// TIA Portal V20 export
DATA_BLOCK "Config"   // DB60
{ DB_Accessible_From_OPC_UA := 'FALSE' }
AUTHOR : ERsystem_FA2_DH. Kim
// stored: Access Published, DBAccessibleFromOPCUA false, DBAccessibleFromWebserver false, MemoryReserve 100, Namespace Unit1.Em4
   VAR RETAIN
      em { ExternalWritable := 'False'} : "LAF_typeEmConfiguration";
      axis { ExternalAccessible := 'False'; ExternalVisible := 'False'; ExternalWritable := 'False'} : Array[1.._.U1EM4_NO_OF_AXES] of DB_ANY;
      cam { ExternalAccessible := 'False'; ExternalVisible := 'False'; ExternalWritable := 'False'} : Array[1.._.U1EM4_NO_OF_CAM] of DB_ANY;
      outputCam { ExternalAccessible := 'False'; ExternalVisible := 'False'; ExternalWritable := 'False'} : Array[1.._.U1EM4_NO_OF_OUTPUTCAM] of DB_ANY;
      cmPnp1stAnodeDetect { S7_SetPoint := 'True'} : "LBC_typeDigitalSignalConfiguration";
      cmPnp2ndAnodeDetect { S7_SetPoint := 'True'} : "LBC_typeDigitalSignalConfiguration";
      cmAnodeAlignTableElectrodeDetect { S7_SetPoint := 'True'} : "LBC_typeDigitalSignalConfiguration";
      cmAnodeNgPnpElectrodeDetect { S7_SetPoint := 'True'} : "LBC_typeDigitalSignalConfiguration";
      cmAnodeNgBoxFullSensorDetect { S7_SetPoint := 'True'} : "LBC_typeDigitalSignalConfiguration";
      cmAnodeNgBoxDetect { S7_SetPoint := 'True'} : "LBC_typeDigitalSignalConfiguration";
      cmAnodeMainPnP1AxisX { ExternalAccessible := 'False'; ExternalVisible := 'False'; ExternalWritable := 'False'} : "LBC_typeAxis64PosConfiguration";
      cmAnodeMainPnP1AxisY { ExternalAccessible := 'False'; ExternalVisible := 'False'; ExternalWritable := 'False'} : "LBC_typeAxis64PosConfiguration";
      cmAnodeMainPnP1AxisZ { ExternalAccessible := 'False'; ExternalVisible := 'False'; ExternalWritable := 'False'} : "LBC_typeAxis64PosConfiguration";
      cmAnodeMainPnP2AxisX { ExternalAccessible := 'False'; ExternalVisible := 'False'; ExternalWritable := 'False'} : "LBC_typeAxis64PosConfiguration";
      cmAnodeMainPnP2AxisZ { ExternalAccessible := 'False'; ExternalVisible := 'False'; ExternalWritable := 'False'} : "LBC_typeAxis64PosConfiguration";
      cmAnodeAlignTableAxisX { ExternalAccessible := 'False'; ExternalVisible := 'False'; ExternalWritable := 'False'} : "LBC_typeAxis64PosConfiguration";
      cmAnodeAlignTableAxisY1 { ExternalAccessible := 'False'; ExternalVisible := 'False'; ExternalWritable := 'False'} : "LBC_typeAxis64PosConfiguration";
      cmAnodeAlignTableAxisY2 { ExternalAccessible := 'False'; ExternalVisible := 'False'; ExternalWritable := 'False'} : "LBC_typeAxis64PosConfiguration";
      cmAnodeMainPnP1RotaryCwCcw { ExternalAccessible := 'False'; ExternalVisible := 'False'; ExternalWritable := 'False'} : "LBC_typeTwoWayActuatorConfiguration";
      cmAnodeMainPnP1SuctionPlateVacuum { ExternalAccessible := 'False'; ExternalVisible := 'False'; ExternalWritable := 'False'} : "LBC_typeTwoWayActuatorConfiguration";
      cmAnodeMainPnP2SuctionPlateVacuum { ExternalAccessible := 'False'; ExternalVisible := 'False'; ExternalWritable := 'False'} : "LBC_typeTwoWayActuatorConfiguration";
      cmAnodeAlignTableSuctionPlateVacuum { ExternalAccessible := 'False'; ExternalVisible := 'False'; ExternalWritable := 'False'} : "LBC_typeTwoWayActuatorConfiguration";
      cmAnodeGlassCleaning { ExternalAccessible := 'False'; ExternalVisible := 'False'; ExternalWritable := 'False'} : "LBC_typeTwoWayActuatorConfiguration";
      cmAnodeNgPnpUpDown { ExternalAccessible := 'False'; ExternalVisible := 'False'; ExternalWritable := 'False'} : "LBC_typeTwoWayActuatorConfiguration";
      cmAnodeNgPnp1stFwdBwd { ExternalAccessible := 'False'; ExternalVisible := 'False'; ExternalWritable := 'False'; S7_SetPoint := 'True'} : "LBC_typeTwoWayActuatorConfiguration";
      cmAnodeNgPnp2ndFwdBwd { ExternalAccessible := 'False'; ExternalVisible := 'False'; ExternalWritable := 'False'; S7_SetPoint := 'True'} : "LBC_typeTwoWayActuatorConfiguration";
      cmAnodeMaintenanceMovingFixFrontRearFwdBwd { ExternalAccessible := 'False'; ExternalVisible := 'False'; ExternalWritable := 'False'} : "LBC_typeTwoWayActuatorConfiguration";
      cmAnodeNgBoxLiftUpDown { ExternalAccessible := 'False'; ExternalVisible := 'False'; ExternalWritable := 'False'; S7_SetPoint := 'True'} : "LBC_typeTwoWayActuatorConfiguration";
      cmAnodeNgBoxLockUpDown { ExternalAccessible := 'False'; ExternalVisible := 'False'; ExternalWritable := 'False'; S7_SetPoint := 'True'} : "LBC_typeTwoWayActuatorConfiguration";
      cmAnodeNgPnpVaccum { ExternalAccessible := 'False'; ExternalVisible := 'False'; ExternalWritable := 'False'; S7_SetPoint := 'True'} : "LBC_typeTwoWayActuatorConfiguration";
      cmAnodeConveyorCoverFwdBwd { S7_SetPoint := 'True'} : "LBC_typeTwoWayActuatorConfiguration";
      cmAnodeConveyorPickUpBlower { S7_SetPoint := 'True'} : "LBC_typeTwoWayActuatorConfiguration";
      cmAnodeVisionControllerInterface { ExternalAccessible := 'False'; ExternalVisible := 'False'; ExternalWritable := 'False'} : "LER_typeVisionConfiguration";
      softCam : Struct
         cmAnodeMainPnP1AxisX : "LER_typeSoftCamInterface";
         cmAnodeMainPnP1AxisY { S7_SetPoint := 'True'} : "LER_typeSoftCamInterface";
         cmAnodeMainPnP1AxisZ { S7_SetPoint := 'True'} : "LER_typeSoftCamInterface";
         cmAnodeMainPnP2AxisX { S7_SetPoint := 'True'} : "LER_typeSoftCamInterface";
         cmAnodeMainPnP2AxisZ { S7_SetPoint := 'True'} : "LER_typeSoftCamInterface";
         cmAnodeAlignTableAxisX { S7_SetPoint := 'True'} : "LER_typeSoftCamInterface";
         cmAnodeAlignTableAxisY1 { S7_SetPoint := 'True'} : "LER_typeSoftCamInterface";
         cmAnodeAlignTableAxisY2 { S7_SetPoint := 'True'} : "LER_typeSoftCamInterface";
      END_STRUCT;
   END_VAR
BEGIN
   em.referenceDesignator.parent := WSTRING#'';
   em.referenceDesignator.relative := WSTRING#'';
   em.referenceDesignator.combined := WSTRING#'';
   axis[1] := 144;   // AnodeMainPnP1AxisX
   axis[2] := 145;   // AnodeMainPnP2AxisX
   axis[3] := 148;   // AnodeMainPnP1AxisY
   axis[4] := 149;   // AnodeMainPnP1AxisZ
   axis[5] := 150;   // AnodeMainPnP2AxisZ
   axis[6] := 154;   // AnodeAlignTableAxisX
   axis[7] := 155;   // AnodeAlignTableAxisY1
   axis[8] := 156;   // AnodeAlignTableAxisY2
   cam[1] := 144;   // AnodeMainPnP1AxisX
   cam[2] := 145;   // AnodeMainPnP2AxisX
   cam[3] := 148;   // AnodeMainPnP1AxisY
   cam[4] := 149;   // AnodeMainPnP1AxisZ
   outputCam[1] := 412;
   outputCam[2] := 413;
   outputCam[3] := 414;
   outputCam[4] := 415;
   outputCam[5] := 441;
   outputCam[6] := 420;
   outputCam[7] := 437;
   outputCam[8] := 438;
   outputCam[9] := 430;
   outputCam[10] := 432;
   outputCam[11] := 436;
   outputCam[12] := 434;
   outputCam[13] := 433;
   outputCam[14] := 431;
   outputCam[15] := 185;
   outputCam[16] := 435;
   outputCam[17] := 442;
   outputCam[18] := 455;
   outputCam[19] := 456;
   outputCam[20] := 134;
   outputCam[21] := 140;
   outputCam[22] := 187;
   cmPnp1stAnodeDetect.referenceDesignator := WSTRING#'Pnp1stAnodeDetect';
   cmPnp1stAnodeDetect.onDelay := T#0MS;
   cmPnp1stAnodeDetect.offDelay := T#0MS;
   cmPnp1stAnodeDetect.default := FALSE;
   cmPnp1stAnodeDetect.invertProcessValue := FALSE;
   cmPnp1stAnodeDetect.disableAlarms := FALSE;
   cmPnp2ndAnodeDetect.referenceDesignator := WSTRING#'Pnp2ndAnodeDetect';
   cmPnp2ndAnodeDetect.onDelay := T#0MS;
   cmPnp2ndAnodeDetect.offDelay := T#0MS;
   cmPnp2ndAnodeDetect.default := FALSE;
   cmPnp2ndAnodeDetect.invertProcessValue := FALSE;
   cmPnp2ndAnodeDetect.disableAlarms := FALSE;
   cmAnodeAlignTableElectrodeDetect.referenceDesignator := WSTRING#'AlignTableElectrodeDetect';
   cmAnodeAlignTableElectrodeDetect.onDelay := T#0MS;
   cmAnodeAlignTableElectrodeDetect.offDelay := T#0MS;
   cmAnodeAlignTableElectrodeDetect.default := FALSE;
   cmAnodeAlignTableElectrodeDetect.invertProcessValue := FALSE;
   cmAnodeAlignTableElectrodeDetect.disableAlarms := FALSE;
   cmAnodeNgPnpElectrodeDetect.referenceDesignator := WSTRING#'NgPnpElectrodeDetect';
   cmAnodeNgPnpElectrodeDetect.onDelay := T#0MS;
   cmAnodeNgPnpElectrodeDetect.offDelay := T#0MS;
   cmAnodeNgPnpElectrodeDetect.default := FALSE;
   cmAnodeNgPnpElectrodeDetect.invertProcessValue := FALSE;
   cmAnodeNgPnpElectrodeDetect.disableAlarms := FALSE;
   cmAnodeNgBoxFullSensorDetect.referenceDesignator := WSTRING#'NgBoxFullSensorDetect';
   cmAnodeNgBoxFullSensorDetect.onDelay := T#0MS;
   cmAnodeNgBoxFullSensorDetect.offDelay := T#0MS;
   cmAnodeNgBoxFullSensorDetect.default := FALSE;
   cmAnodeNgBoxFullSensorDetect.invertProcessValue := FALSE;
   cmAnodeNgBoxFullSensorDetect.disableAlarms := FALSE;
   cmAnodeNgBoxDetect.referenceDesignator := WSTRING#'NgBoxDetect';
   cmAnodeNgBoxDetect.onDelay := T#0MS;
   cmAnodeNgBoxDetect.offDelay := T#0MS;
   cmAnodeNgBoxDetect.default := FALSE;
   cmAnodeNgBoxDetect.invertProcessValue := FALSE;
   cmAnodeNgBoxDetect.disableAlarms := FALSE;
   cmAnodeMainPnP1AxisX.referenceDesignator := WSTRING#'AnodeMainPnP1AxisX';
   cmAnodeMainPnP1AxisX.disableAlarms := FALSE;
   cmAnodeMainPnP1AxisX.masterControlPopUp := TRUE;
   cmAnodeMainPnP1AxisX.setPositions[0].position := 540.0;
   cmAnodeMainPnP1AxisX.setPositions[1].position := 0.0;
   cmAnodeMainPnP1AxisX.setPositions[2].position := -5.0;
   cmAnodeMainPnP1AxisX.setPositions[3..15].position := 0.0;
   cmAnodeMainPnP1AxisX.setPositions[0..1].velocity := 500.0;
   cmAnodeMainPnP1AxisX.setPositions[2..3].velocity := 1040.0;
   cmAnodeMainPnP1AxisX.setPositions[4..15].velocity := -1.0;
   cmAnodeMainPnP1AxisX.setPositions[0..1].acceleration := 5000.0;
   cmAnodeMainPnP1AxisX.setPositions[2..3].acceleration := 10400.0;
   cmAnodeMainPnP1AxisX.setPositions[4..15].acceleration := -1.0;
   cmAnodeMainPnP1AxisX.setPositions[0..1].deceleration := 5000.0;
   cmAnodeMainPnP1AxisX.setPositions[2..3].deceleration := 10400.0;
   cmAnodeMainPnP1AxisX.setPositions[4..15].deceleration := -1.0;
   cmAnodeMainPnP1AxisX.setPositions[0..15]."name" := '';
   cmAnodeMainPnP1AxisY.referenceDesignator := WSTRING#'AnodeMainPnP1AxisY';
   cmAnodeMainPnP1AxisY.disableAlarms := FALSE;
   cmAnodeMainPnP1AxisY.masterControlPopUp := TRUE;
   cmAnodeMainPnP1AxisY.setPositions[0..15].position := 0.0;
   cmAnodeMainPnP1AxisY.setPositions[0].velocity := 50.0;
   cmAnodeMainPnP1AxisY.setPositions[1].velocity := 30.0;
   cmAnodeMainPnP1AxisY.setPositions[2..15].velocity := -1.0;
   cmAnodeMainPnP1AxisY.setPositions[0].acceleration := 500.0;
   cmAnodeMainPnP1AxisY.setPositions[1].acceleration := 30.0;
   cmAnodeMainPnP1AxisY.setPositions[2..15].acceleration := -1.0;
   cmAnodeMainPnP1AxisY.setPositions[0].deceleration := 500.0;
   cmAnodeMainPnP1AxisY.setPositions[1].deceleration := 30.0;
   cmAnodeMainPnP1AxisY.setPositions[2..15].deceleration := -1.0;
   cmAnodeMainPnP1AxisY.setPositions[0..15]."name" := '';
   cmAnodeMainPnP1AxisZ.referenceDesignator := WSTRING#'AnodeMainPnP1AxisZ';
   cmAnodeMainPnP1AxisZ.disableAlarms := FALSE;
   cmAnodeMainPnP1AxisZ.masterControlPopUp := TRUE;
   cmAnodeMainPnP1AxisZ.setPositions[0].position := 0.0;
   cmAnodeMainPnP1AxisZ.setPositions[1].position := 20.0;
   cmAnodeMainPnP1AxisZ.setPositions[2..3].position := 30.0;
   cmAnodeMainPnP1AxisZ.setPositions[4..15].position := 0.0;
   cmAnodeMainPnP1AxisZ.setPositions[0..3].velocity := 50.0;
   cmAnodeMainPnP1AxisZ.setPositions[4..15].velocity := -1.0;
   cmAnodeMainPnP1AxisZ.setPositions[0..3].acceleration := 500.0;
   cmAnodeMainPnP1AxisZ.setPositions[4..15].acceleration := -1.0;
   cmAnodeMainPnP1AxisZ.setPositions[0..3].deceleration := 500.0;
   cmAnodeMainPnP1AxisZ.setPositions[4..15].deceleration := -1.0;
   cmAnodeMainPnP1AxisZ.setPositions[0..15]."name" := '';
   cmAnodeMainPnP2AxisX.referenceDesignator := WSTRING#'AnodeMainPnP2AxisX';
   cmAnodeMainPnP2AxisX.disableAlarms := FALSE;
   cmAnodeMainPnP2AxisX.masterControlPopUp := TRUE;
   cmAnodeMainPnP2AxisX.setPositions[0].position := 540.0;
   cmAnodeMainPnP2AxisX.setPositions[1].position := 0.0;
   cmAnodeMainPnP2AxisX.setPositions[2].position := -3.5;
   cmAnodeMainPnP2AxisX.setPositions[3..15].position := 0.0;
   cmAnodeMainPnP2AxisX.setPositions[0..1].velocity := 500.0;
   cmAnodeMainPnP2AxisX.setPositions[2..3].velocity := 1040.0;
   cmAnodeMainPnP2AxisX.setPositions[4..15].velocity := -1.0;
   cmAnodeMainPnP2AxisX.setPositions[0..1].acceleration := 5000.0;
   cmAnodeMainPnP2AxisX.setPositions[2..3].acceleration := 10400.0;
   cmAnodeMainPnP2AxisX.setPositions[4..15].acceleration := -1.0;
   cmAnodeMainPnP2AxisX.setPositions[0..1].deceleration := 5000.0;
   cmAnodeMainPnP2AxisX.setPositions[2..3].deceleration := 10400.0;
   cmAnodeMainPnP2AxisX.setPositions[4..15].deceleration := -1.0;
   cmAnodeMainPnP2AxisX.setPositions[0..15]."name" := '';
   cmAnodeMainPnP2AxisZ.referenceDesignator := WSTRING#'AnodeMainPnP2AxisZ';
   cmAnodeMainPnP2AxisZ.disableAlarms := FALSE;
   cmAnodeMainPnP2AxisZ.masterControlPopUp := TRUE;
   cmAnodeMainPnP2AxisZ.setPositions[0].position := 0.0;
   cmAnodeMainPnP2AxisZ.setPositions[1].position := 20.0;
   cmAnodeMainPnP2AxisZ.setPositions[2..3].position := 30.0;
   cmAnodeMainPnP2AxisZ.setPositions[4..15].position := 0.0;
   cmAnodeMainPnP2AxisZ.setPositions[0..3].velocity := 50.0;
   cmAnodeMainPnP2AxisZ.setPositions[4..15].velocity := -1.0;
   cmAnodeMainPnP2AxisZ.setPositions[0..3].acceleration := 500.0;
   cmAnodeMainPnP2AxisZ.setPositions[4..15].acceleration := -1.0;
   cmAnodeMainPnP2AxisZ.setPositions[0..3].deceleration := 500.0;
   cmAnodeMainPnP2AxisZ.setPositions[4..15].deceleration := -1.0;
   cmAnodeMainPnP2AxisZ.setPositions[0..15]."name" := '';
   cmAnodeAlignTableAxisX.referenceDesignator := WSTRING#'AnodeAlignTableAxisX';
   cmAnodeAlignTableAxisX.disableAlarms := FALSE;
   cmAnodeAlignTableAxisX.masterControlPopUp := TRUE;
   cmAnodeAlignTableAxisX.setPositions[0].position := 0.0;
   cmAnodeAlignTableAxisX.setPositions[1].position := 1.0;
   cmAnodeAlignTableAxisX.setPositions[2..3].position := -4.08;
   cmAnodeAlignTableAxisX.setPositions[4].position := -2.08;
   cmAnodeAlignTableAxisX.setPositions[5..7].position := -0.08;
   cmAnodeAlignTableAxisX.setPositions[8].position := -2.08;
   cmAnodeAlignTableAxisX.setPositions[9].position := -4.08;
   cmAnodeAlignTableAxisX.setPositions[10].position := 8.5;
   cmAnodeAlignTableAxisX.setPositions[11..15].position := 0.0;
   cmAnodeAlignTableAxisX.setPositions[0..1].velocity := 50.0;
   cmAnodeAlignTableAxisX.setPositions[2..9].velocity := 30.0;
   cmAnodeAlignTableAxisX.setPositions[10..15].velocity := -1.0;
   cmAnodeAlignTableAxisX.setPositions[0..1].acceleration := 500.0;
   cmAnodeAlignTableAxisX.setPositions[2..9].acceleration := 30.0;
   cmAnodeAlignTableAxisX.setPositions[10..15].acceleration := -1.0;
   cmAnodeAlignTableAxisX.setPositions[0..1].deceleration := 500.0;
   cmAnodeAlignTableAxisX.setPositions[2..9].deceleration := 30.0;
   cmAnodeAlignTableAxisX.setPositions[10..15].deceleration := -1.0;
   cmAnodeAlignTableAxisX.setPositions[0..15]."name" := '';
   cmAnodeAlignTableAxisY1.referenceDesignator := WSTRING#'AnodeAlignTableAxisY1';
   cmAnodeAlignTableAxisY1.disableAlarms := FALSE;
   cmAnodeAlignTableAxisY1.masterControlPopUp := TRUE;
   cmAnodeAlignTableAxisY1.setPositions[0].position := 0.0;
   cmAnodeAlignTableAxisY1.setPositions[1].position := 2.0;
   cmAnodeAlignTableAxisY1.setPositions[2].position := 0.6;
   cmAnodeAlignTableAxisY1.setPositions[3..5].position := 2.6;
   cmAnodeAlignTableAxisY1.setPositions[6].position := 0.6;
   cmAnodeAlignTableAxisY1.setPositions[7].position := -1.4;
   cmAnodeAlignTableAxisY1.setPositions[8].position := 0.6;
   cmAnodeAlignTableAxisY1.setPositions[9].position := -1.4;
   cmAnodeAlignTableAxisY1.setPositions[10].position := 8.5;
   cmAnodeAlignTableAxisY1.setPositions[11..15].position := 0.0;
   cmAnodeAlignTableAxisY1.setPositions[0..1].velocity := 50.0;
   cmAnodeAlignTableAxisY1.setPositions[2..9].velocity := 30.0;
   cmAnodeAlignTableAxisY1.setPositions[10..15].velocity := -1.0;
   cmAnodeAlignTableAxisY1.setPositions[0..1].acceleration := 500.0;
   cmAnodeAlignTableAxisY1.setPositions[2..9].acceleration := 30.0;
   cmAnodeAlignTableAxisY1.setPositions[10..15].acceleration := -1.0;
   cmAnodeAlignTableAxisY1.setPositions[0..1].deceleration := 500.0;
   cmAnodeAlignTableAxisY1.setPositions[2..9].deceleration := 30.0;
   cmAnodeAlignTableAxisY1.setPositions[10..15].deceleration := -1.0;
   cmAnodeAlignTableAxisY1.setPositions[0..15]."name" := '';
   cmAnodeAlignTableAxisY2.referenceDesignator := WSTRING#'AnodeAlignTableAxisY2';
   cmAnodeAlignTableAxisY2.disableAlarms := FALSE;
   cmAnodeAlignTableAxisY2.masterControlPopUp := TRUE;
   cmAnodeAlignTableAxisY2.setPositions[0].position := 0.0;
   cmAnodeAlignTableAxisY2.setPositions[1].position := 3.0;
   cmAnodeAlignTableAxisY2.setPositions[2..9].position := 0.0;
   cmAnodeAlignTableAxisY2.setPositions[10].position := 8.5;
   cmAnodeAlignTableAxisY2.setPositions[11..15].position := 0.0;
   cmAnodeAlignTableAxisY2.setPositions[0..1].velocity := 50.0;
   cmAnodeAlignTableAxisY2.setPositions[2..15].velocity := -1.0;
   cmAnodeAlignTableAxisY2.setPositions[0..1].acceleration := 500.0;
   cmAnodeAlignTableAxisY2.setPositions[2..15].acceleration := -1.0;
   cmAnodeAlignTableAxisY2.setPositions[0..1].deceleration := 500.0;
   cmAnodeAlignTableAxisY2.setPositions[2..15].deceleration := -1.0;
   cmAnodeAlignTableAxisY2.setPositions[0..15]."name" := '';
   cmAnodeMainPnP1RotaryCwCcw.monitoringLeavingFeedback := T#1S;
   cmAnodeMainPnP1RotaryCwCcw.monitoringReachingFeedback := T#1S;
   cmAnodeMainPnP1RotaryCwCcw.monitoringDiscrepancy := T#0MS;
   cmAnodeMainPnP1RotaryCwCcw.setOutputHomeContinuously := TRUE;
   cmAnodeMainPnP1RotaryCwCcw.setOutputWorkContinuously := TRUE;
   cmAnodeMainPnP1RotaryCwCcw.disableHomeCommand := FALSE;
   cmAnodeMainPnP1RotaryCwCcw.disableFeedbackHomePos := TRUE;
   cmAnodeMainPnP1RotaryCwCcw.disableFeedbackWorkPos := TRUE;
   cmAnodeMainPnP1RotaryCwCcw.disableAlarms := TRUE;
   cmAnodeMainPnP1RotaryCwCcw.resetOutputsOnError := FALSE;
   cmAnodeMainPnP1RotaryCwCcw.allwaysWaitOnReachingTime := FALSE;
   cmAnodeMainPnP1SuctionPlateVacuum.monitoringLeavingFeedback := T#1S;
   cmAnodeMainPnP1SuctionPlateVacuum.monitoringReachingFeedback := T#1S;
   cmAnodeMainPnP1SuctionPlateVacuum.monitoringDiscrepancy := T#15S;
   cmAnodeMainPnP1SuctionPlateVacuum.setOutputHomeContinuously := TRUE;
   cmAnodeMainPnP1SuctionPlateVacuum.setOutputWorkContinuously := TRUE;
   cmAnodeMainPnP1SuctionPlateVacuum.disableHomeCommand := FALSE;
   cmAnodeMainPnP1SuctionPlateVacuum.disableFeedbackHomePos := FALSE;
   cmAnodeMainPnP1SuctionPlateVacuum.disableFeedbackWorkPos := FALSE;
   cmAnodeMainPnP1SuctionPlateVacuum.disableAlarms := FALSE;
   cmAnodeMainPnP1SuctionPlateVacuum.resetOutputsOnError := FALSE;
   cmAnodeMainPnP1SuctionPlateVacuum.allwaysWaitOnReachingTime := FALSE;
   cmAnodeMainPnP2SuctionPlateVacuum.monitoringLeavingFeedback := T#1S;
   cmAnodeMainPnP2SuctionPlateVacuum.monitoringReachingFeedback := T#1S;
   cmAnodeMainPnP2SuctionPlateVacuum.monitoringDiscrepancy := T#15S;
   cmAnodeMainPnP2SuctionPlateVacuum.setOutputHomeContinuously := TRUE;
   cmAnodeMainPnP2SuctionPlateVacuum.setOutputWorkContinuously := TRUE;
   cmAnodeMainPnP2SuctionPlateVacuum.disableHomeCommand := FALSE;
   cmAnodeMainPnP2SuctionPlateVacuum.disableFeedbackHomePos := FALSE;
   cmAnodeMainPnP2SuctionPlateVacuum.disableFeedbackWorkPos := FALSE;
   cmAnodeMainPnP2SuctionPlateVacuum.disableAlarms := FALSE;
   cmAnodeMainPnP2SuctionPlateVacuum.resetOutputsOnError := FALSE;
   cmAnodeMainPnP2SuctionPlateVacuum.allwaysWaitOnReachingTime := FALSE;
   cmAnodeAlignTableSuctionPlateVacuum.monitoringLeavingFeedback := T#1S;
   cmAnodeAlignTableSuctionPlateVacuum.monitoringReachingFeedback := T#1S;
   cmAnodeAlignTableSuctionPlateVacuum.monitoringDiscrepancy := T#0MS;
   cmAnodeAlignTableSuctionPlateVacuum.setOutputHomeContinuously := TRUE;
   cmAnodeAlignTableSuctionPlateVacuum.setOutputWorkContinuously := TRUE;
   cmAnodeAlignTableSuctionPlateVacuum.disableHomeCommand := FALSE;
   cmAnodeAlignTableSuctionPlateVacuum.disableFeedbackHomePos := FALSE;
   cmAnodeAlignTableSuctionPlateVacuum.disableFeedbackWorkPos := FALSE;
   cmAnodeAlignTableSuctionPlateVacuum.disableAlarms := FALSE;
   cmAnodeAlignTableSuctionPlateVacuum.resetOutputsOnError := FALSE;
   cmAnodeAlignTableSuctionPlateVacuum.allwaysWaitOnReachingTime := FALSE;
   cmAnodeGlassCleaning.monitoringLeavingFeedback := T#1S;
   cmAnodeGlassCleaning.monitoringReachingFeedback := T#1S;
   cmAnodeGlassCleaning.monitoringDiscrepancy := T#0MS;
   cmAnodeGlassCleaning.setOutputHomeContinuously := TRUE;
   cmAnodeGlassCleaning.setOutputWorkContinuously := TRUE;
   cmAnodeGlassCleaning.disableHomeCommand := FALSE;
   cmAnodeGlassCleaning.disableFeedbackHomePos := TRUE;
   cmAnodeGlassCleaning.disableFeedbackWorkPos := TRUE;
   cmAnodeGlassCleaning.disableAlarms := FALSE;
   cmAnodeGlassCleaning.resetOutputsOnError := FALSE;
   cmAnodeGlassCleaning.allwaysWaitOnReachingTime := FALSE;
   cmAnodeNgPnpUpDown.monitoringLeavingFeedback := T#5S;
   cmAnodeNgPnpUpDown.monitoringReachingFeedback := T#5S;
   cmAnodeNgPnpUpDown.monitoringDiscrepancy := T#0MS;
   cmAnodeNgPnpUpDown.setOutputHomeContinuously := TRUE;
   cmAnodeNgPnpUpDown.setOutputWorkContinuously := TRUE;
   cmAnodeNgPnpUpDown.disableHomeCommand := FALSE;
   cmAnodeNgPnpUpDown.disableFeedbackHomePos := TRUE;
   cmAnodeNgPnpUpDown.disableFeedbackWorkPos := TRUE;
   cmAnodeNgPnpUpDown.disableAlarms := FALSE;
   cmAnodeNgPnpUpDown.resetOutputsOnError := FALSE;
   cmAnodeNgPnpUpDown.allwaysWaitOnReachingTime := FALSE;
   cmAnodeNgPnp1stFwdBwd.monitoringLeavingFeedback := T#5S;
   cmAnodeNgPnp1stFwdBwd.monitoringReachingFeedback := T#5S;
   cmAnodeNgPnp1stFwdBwd.monitoringDiscrepancy := T#0MS;
   cmAnodeNgPnp1stFwdBwd.setOutputHomeContinuously := TRUE;
   cmAnodeNgPnp1stFwdBwd.setOutputWorkContinuously := TRUE;
   cmAnodeNgPnp1stFwdBwd.disableHomeCommand := FALSE;
   cmAnodeNgPnp1stFwdBwd.disableFeedbackHomePos := TRUE;
   cmAnodeNgPnp1stFwdBwd.disableFeedbackWorkPos := TRUE;
   cmAnodeNgPnp1stFwdBwd.disableAlarms := FALSE;
   cmAnodeNgPnp1stFwdBwd.resetOutputsOnError := FALSE;
   cmAnodeNgPnp1stFwdBwd.allwaysWaitOnReachingTime := FALSE;
   cmAnodeNgPnp2ndFwdBwd.monitoringLeavingFeedback := T#0MS;
   cmAnodeNgPnp2ndFwdBwd.monitoringReachingFeedback := T#0MS;
   cmAnodeNgPnp2ndFwdBwd.monitoringDiscrepancy := T#0MS;
   cmAnodeNgPnp2ndFwdBwd.setOutputHomeContinuously := FALSE;
   cmAnodeNgPnp2ndFwdBwd.setOutputWorkContinuously := FALSE;
   cmAnodeNgPnp2ndFwdBwd.disableHomeCommand := FALSE;
   cmAnodeNgPnp2ndFwdBwd.disableFeedbackHomePos := TRUE;
   cmAnodeNgPnp2ndFwdBwd.disableFeedbackWorkPos := TRUE;
   cmAnodeNgPnp2ndFwdBwd.disableAlarms := FALSE;
   cmAnodeNgPnp2ndFwdBwd.resetOutputsOnError := FALSE;
   cmAnodeNgPnp2ndFwdBwd.allwaysWaitOnReachingTime := FALSE;
   cmAnodeMaintenanceMovingFixFrontRearFwdBwd.monitoringLeavingFeedback := T#5S;
   cmAnodeMaintenanceMovingFixFrontRearFwdBwd.monitoringReachingFeedback := T#5S;
   cmAnodeMaintenanceMovingFixFrontRearFwdBwd.monitoringDiscrepancy := T#0MS;
   cmAnodeMaintenanceMovingFixFrontRearFwdBwd.setOutputHomeContinuously := TRUE;
   cmAnodeMaintenanceMovingFixFrontRearFwdBwd.setOutputWorkContinuously := TRUE;
   cmAnodeMaintenanceMovingFixFrontRearFwdBwd.disableHomeCommand := FALSE;
   cmAnodeMaintenanceMovingFixFrontRearFwdBwd.disableFeedbackHomePos := TRUE;
   cmAnodeMaintenanceMovingFixFrontRearFwdBwd.disableFeedbackWorkPos := TRUE;
   cmAnodeMaintenanceMovingFixFrontRearFwdBwd.disableAlarms := FALSE;
   cmAnodeMaintenanceMovingFixFrontRearFwdBwd.resetOutputsOnError := FALSE;
   cmAnodeMaintenanceMovingFixFrontRearFwdBwd.allwaysWaitOnReachingTime := FALSE;
   cmAnodeNgBoxLiftUpDown.monitoringLeavingFeedback := T#5S;
   cmAnodeNgBoxLiftUpDown.monitoringReachingFeedback := T#5S;
   cmAnodeNgBoxLiftUpDown.monitoringDiscrepancy := T#0MS;
   cmAnodeNgBoxLiftUpDown.setOutputHomeContinuously := TRUE;
   cmAnodeNgBoxLiftUpDown.setOutputWorkContinuously := TRUE;
   cmAnodeNgBoxLiftUpDown.disableHomeCommand := FALSE;
   cmAnodeNgBoxLiftUpDown.disableFeedbackHomePos := TRUE;
   cmAnodeNgBoxLiftUpDown.disableFeedbackWorkPos := TRUE;
   cmAnodeNgBoxLiftUpDown.disableAlarms := FALSE;
   cmAnodeNgBoxLiftUpDown.resetOutputsOnError := FALSE;
   cmAnodeNgBoxLiftUpDown.allwaysWaitOnReachingTime := FALSE;
   cmAnodeNgBoxLockUpDown.monitoringLeavingFeedback := T#5S;
   cmAnodeNgBoxLockUpDown.monitoringReachingFeedback := T#5S;
   cmAnodeNgBoxLockUpDown.monitoringDiscrepancy := T#0MS;
   cmAnodeNgBoxLockUpDown.setOutputHomeContinuously := TRUE;
   cmAnodeNgBoxLockUpDown.setOutputWorkContinuously := TRUE;
   cmAnodeNgBoxLockUpDown.disableHomeCommand := FALSE;
   cmAnodeNgBoxLockUpDown.disableFeedbackHomePos := FALSE;
   cmAnodeNgBoxLockUpDown.disableFeedbackWorkPos := FALSE;
   cmAnodeNgBoxLockUpDown.disableAlarms := FALSE;
   cmAnodeNgBoxLockUpDown.resetOutputsOnError := FALSE;
   cmAnodeNgBoxLockUpDown.allwaysWaitOnReachingTime := FALSE;
   cmAnodeNgPnpVaccum.monitoringLeavingFeedback := T#5S;
   cmAnodeNgPnpVaccum.monitoringReachingFeedback := T#5S;
   cmAnodeNgPnpVaccum.monitoringDiscrepancy := T#0MS;
   cmAnodeNgPnpVaccum.setOutputHomeContinuously := TRUE;
   cmAnodeNgPnpVaccum.setOutputWorkContinuously := TRUE;
   cmAnodeNgPnpVaccum.disableHomeCommand := FALSE;
   cmAnodeNgPnpVaccum.disableFeedbackHomePos := FALSE;
   cmAnodeNgPnpVaccum.disableFeedbackWorkPos := FALSE;
   cmAnodeNgPnpVaccum.disableAlarms := FALSE;
   cmAnodeNgPnpVaccum.resetOutputsOnError := FALSE;
   cmAnodeNgPnpVaccum.allwaysWaitOnReachingTime := FALSE;
   cmAnodeConveyorCoverFwdBwd.monitoringLeavingFeedback := T#5S;
   cmAnodeConveyorCoverFwdBwd.monitoringReachingFeedback := T#5S;
   cmAnodeConveyorCoverFwdBwd.monitoringDiscrepancy := T#0MS;
   cmAnodeConveyorCoverFwdBwd.setOutputHomeContinuously := TRUE;
   cmAnodeConveyorCoverFwdBwd.setOutputWorkContinuously := TRUE;
   cmAnodeConveyorCoverFwdBwd.disableHomeCommand := FALSE;
   cmAnodeConveyorCoverFwdBwd.disableFeedbackHomePos := TRUE;
   cmAnodeConveyorCoverFwdBwd.disableFeedbackWorkPos := TRUE;
   cmAnodeConveyorCoverFwdBwd.disableAlarms := FALSE;
   cmAnodeConveyorCoverFwdBwd.resetOutputsOnError := FALSE;
   cmAnodeConveyorCoverFwdBwd.allwaysWaitOnReachingTime := FALSE;
   cmAnodeConveyorPickUpBlower.monitoringLeavingFeedback := T#0MS;
   cmAnodeConveyorPickUpBlower.monitoringReachingFeedback := T#0MS;
   cmAnodeConveyorPickUpBlower.monitoringDiscrepancy := T#0MS;
   cmAnodeConveyorPickUpBlower.setOutputHomeContinuously := TRUE;
   cmAnodeConveyorPickUpBlower.setOutputWorkContinuously := TRUE;
   cmAnodeConveyorPickUpBlower.disableHomeCommand := FALSE;
   cmAnodeConveyorPickUpBlower.disableFeedbackHomePos := TRUE;
   cmAnodeConveyorPickUpBlower.disableFeedbackWorkPos := TRUE;
   cmAnodeConveyorPickUpBlower.disableAlarms := FALSE;
   cmAnodeConveyorPickUpBlower.resetOutputsOnError := FALSE;
   cmAnodeConveyorPickUpBlower.allwaysWaitOnReachingTime := FALSE;
   cmAnodeVisionControllerInterface.hwID.cmdResultStatusID := 394;
   cmAnodeVisionControllerInterface.hwID.trgReadyStatusID := 395;
   cmAnodeVisionControllerInterface.hwID.trgAckStatusID := 396;
   cmAnodeVisionControllerInterface.hwID.miscellaneousStatusID := 397;
   cmAnodeVisionControllerInterface.hwID.assignableStatusID := 398;
   cmAnodeVisionControllerInterface.hwID.resultData248ByteID_1 := 399;
   cmAnodeVisionControllerInterface.hwID.resultData248ByteID_2 := 578;
   cmAnodeVisionControllerInterface.hwID.resultData248ByteID_3 := 579;
   cmAnodeVisionControllerInterface.hwID.resultData248ByteID_4 := 581;
   cmAnodeVisionControllerInterface.hwID.resultData248ByteID_5 := 582;
   cmAnodeVisionControllerInterface.hwID.cmdResultControlID := 400;
   cmAnodeVisionControllerInterface.hwID.trgControlID := 401;
   cmAnodeVisionControllerInterface.hwID.miscellaneousControlID := 402;
   cmAnodeVisionControllerInterface.hwID.reservedControlID := 403;
   cmAnodeVisionControllerInterface.hwID.assignableControlID := 404;
   cmAnodeVisionControllerInterface.hwID.parameterData248ByteID_1 := 405;
   cmAnodeVisionControllerInterface.hwID.parameterData248ByteID_2 := 681;
   cmAnodeVisionControllerInterface.hwID.parameterData248ByteID_3 := 718;
   cmAnodeVisionControllerInterface.hwID.parameterData248ByteID_4 := 832;
   cmAnodeVisionControllerInterface.hwID.parameterData248ByteID_5 := 841;
   cmAnodeVisionControllerInterface.referenceDesignator := WSTRING#'VisionControllerInterface';
   cmAnodeVisionControllerInterface.disableAlarms := FALSE;
   cmAnodeVisionControllerInterface.trigger1Use := FALSE;
   cmAnodeVisionControllerInterface.trigger2Use := FALSE;
   cmAnodeVisionControllerInterface.trigger3Use := FALSE;
   cmAnodeVisionControllerInterface.trigger4Use := FALSE;
   cmAnodeVisionControllerInterface.triggertime := T#0MS;
   cmAnodeVisionControllerInterface.cycleTime := T#0MS;
   cmAnodeVisionControllerInterface.DataConfig.cmdResultControl.cmdRequest := FALSE;
   cmAnodeVisionControllerInterface.DataConfig.cmdResultControl.inDataFbSyncInhibit := FALSE;
   cmAnodeVisionControllerInterface.DataConfig.cmdResultControl.reserved := FALSE;
   cmAnodeVisionControllerInterface.DataConfig.cmdResultControl.resultAck := FALSE;
   cmAnodeVisionControllerInterface.DataConfig.cmdResultControl.err0ResetRequest := FALSE;
   cmAnodeVisionControllerInterface.DataConfig.cmdResultControl.err1ResetRequest := FALSE;
   cmAnodeVisionControllerInterface.DataConfig.cmdResultControl.reserved0 := FALSE;
   cmAnodeVisionControllerInterface.DataConfig.cmdResultControl.reserved1 := FALSE;
   cmAnodeVisionControllerInterface.DataConfig.trgControl.trg1 := FALSE;
   cmAnodeVisionControllerInterface.DataConfig.trgControl.trg2 := FALSE;
   cmAnodeVisionControllerInterface.DataConfig.trgControl.trg3 := FALSE;
   cmAnodeVisionControllerInterface.DataConfig.trgControl.trg4 := FALSE;
   cmAnodeVisionControllerInterface.DataConfig.trgControl.reserved0 := FALSE;
   cmAnodeVisionControllerInterface.DataConfig.trgControl.reserved1 := FALSE;
   cmAnodeVisionControllerInterface.DataConfig.trgControl.reserved2 := FALSE;
   cmAnodeVisionControllerInterface.DataConfig.trgControl.reserved3 := FALSE;
   cmAnodeVisionControllerInterface.DataConfig.miscellaneousControl.reset := FALSE;
   cmAnodeVisionControllerInterface.DataConfig.miscellaneousControl.ext := FALSE;
   cmAnodeVisionControllerInterface.DataConfig.miscellaneousControl.test := FALSE;
   cmAnodeVisionControllerInterface.DataConfig.miscellaneousControl.reserved0 := FALSE;
   cmAnodeVisionControllerInterface.DataConfig.miscellaneousControl.reserved1 := FALSE;
   cmAnodeVisionControllerInterface.DataConfig.miscellaneousControl.reserved2 := FALSE;
   cmAnodeVisionControllerInterface.DataConfig.miscellaneousControl.reserved3 := FALSE;
   cmAnodeVisionControllerInterface.DataConfig.miscellaneousControl.reserved4 := FALSE;
   cmAnodeVisionControllerInterface.DataConfig.reservedControl.reserved0 := FALSE;
   cmAnodeVisionControllerInterface.DataConfig.reservedControl.reserved1 := FALSE;
   cmAnodeVisionControllerInterface.DataConfig.reservedControl.reserved2 := FALSE;
   cmAnodeVisionControllerInterface.DataConfig.reservedControl.reserved3 := FALSE;
   cmAnodeVisionControllerInterface.DataConfig.reservedControl.reserved4 := FALSE;
   cmAnodeVisionControllerInterface.DataConfig.reservedControl.reserved5 := FALSE;
   cmAnodeVisionControllerInterface.DataConfig.reservedControl.reserved6 := FALSE;
   cmAnodeVisionControllerInterface.DataConfig.reservedControl.reserved7 := FALSE;
   cmAnodeVisionControllerInterface.DataConfig.assignableControl.assignable_0 := FALSE;
   cmAnodeVisionControllerInterface.DataConfig.assignableControl.assignable_1 := FALSE;
   cmAnodeVisionControllerInterface.DataConfig.assignableControl.assignable_2 := FALSE;
   cmAnodeVisionControllerInterface.DataConfig.assignableControl.assignable_3 := FALSE;
   cmAnodeVisionControllerInterface.DataConfig.assignableControl.assignable_4 := FALSE;
   cmAnodeVisionControllerInterface.DataConfig.assignableControl.assignable_5 := FALSE;
   cmAnodeVisionControllerInterface.DataConfig.assignableControl.assignable_6 := FALSE;
   cmAnodeVisionControllerInterface.DataConfig.assignableControl.assignable_7 := FALSE;
   cmAnodeVisionControllerInterface.DataConfig.assignableControl.assignable_8 := FALSE;
   cmAnodeVisionControllerInterface.DataConfig.assignableControl.assignable_9 := FALSE;
   cmAnodeVisionControllerInterface.DataConfig.assignableControl.assignable_10 := FALSE;
   cmAnodeVisionControllerInterface.DataConfig.assignableControl.assignable_11 := FALSE;
   cmAnodeVisionControllerInterface.DataConfig.assignableControl.assignable_12 := FALSE;
   cmAnodeVisionControllerInterface.DataConfig.assignableControl.assignable_13 := FALSE;
   cmAnodeVisionControllerInterface.DataConfig.assignableControl.assignable_14 := FALSE;
   cmAnodeVisionControllerInterface.DataConfig.assignableControl.assignable_15 := FALSE;
   cmAnodeVisionControllerInterface.DataConfig.assignableControl.assignable_16 := FALSE;
   cmAnodeVisionControllerInterface.DataConfig.assignableControl.assignable_17 := FALSE;
   cmAnodeVisionControllerInterface.DataConfig.assignableControl.assignable_18 := FALSE;
   cmAnodeVisionControllerInterface.DataConfig.assignableControl.assignable_19 := FALSE;
   cmAnodeVisionControllerInterface.DataConfig.assignableControl.assignable_20 := FALSE;
   cmAnodeVisionControllerInterface.DataConfig.assignableControl.assignable_21 := FALSE;
   cmAnodeVisionControllerInterface.DataConfig.assignableControl.assignable_22 := FALSE;
   cmAnodeVisionControllerInterface.DataConfig.assignableControl.assignable_23 := FALSE;
   cmAnodeVisionControllerInterface.DataConfig.assignableControl.assignable_24 := FALSE;
   cmAnodeVisionControllerInterface.DataConfig.assignableControl.assignable_25 := FALSE;
   cmAnodeVisionControllerInterface.DataConfig.assignableControl.assignable_26 := FALSE;
   cmAnodeVisionControllerInterface.DataConfig.assignableControl.assignable_27 := FALSE;
   cmAnodeVisionControllerInterface.DataConfig.assignableControl.assignable_28 := FALSE;
   cmAnodeVisionControllerInterface.DataConfig.assignableControl.assignable_29 := FALSE;
   cmAnodeVisionControllerInterface.DataConfig.assignableControl.assignable_30 := FALSE;
   cmAnodeVisionControllerInterface.DataConfig.assignableControl.assignable_31 := FALSE;
   cmAnodeVisionControllerInterface.DataConfig.parameterData248Byte_1.reversed0 := 0;
   cmAnodeVisionControllerInterface.DataConfig.parameterData248Byte_1.reserved1 := 0;
   cmAnodeVisionControllerInterface.DataConfig.parameterData248Byte_1.commandNumber := 0;
   cmAnodeVisionControllerInterface.DataConfig.parameterData248Byte_1.cmdParameter[0..15] := 0;
   cmAnodeVisionControllerInterface.DataConfig.parameterData248Byte_1.inDataFieldbus[0..42] := 0;
   cmAnodeVisionControllerInterface.DataConfig.parameterData248Byte_2[0..61] := 0;
   cmAnodeVisionControllerInterface.DataConfig.parameterData248Byte_3[0..61] := 0;
   cmAnodeVisionControllerInterface.DataConfig.parameterData248Byte_4[0..61] := 0;
   cmAnodeVisionControllerInterface.DataConfig.parameterData248Byte_5[0..61] := 0;
   softCam.cmAnodeMainPnP1AxisX.TargetPosition := 0.0;
   softCam.cmAnodeMainPnP1AxisX.ActualPosition := 0.0;
   softCam.cmAnodeMainPnP1AxisX.UnitName := WSTRING#'';
   softCam.cmAnodeMainPnP1AxisX.error := FALSE;
   softCam.cmAnodeMainPnP1AxisX.status := 16#0000;
   softCam.cmAnodeMainPnP1AxisX.position[0..15].SetValue.Negative := 0.0;
   softCam.cmAnodeMainPnP1AxisX.position[0..15].SetValue.Postive := 0.0;
   softCam.cmAnodeMainPnP1AxisX.position[0..15].ProcessValue.Postive := 0.0;
   softCam.cmAnodeMainPnP1AxisX.position[0..15].ProcessValue.Negative := 0.0;
   softCam.cmAnodeMainPnP1AxisX.position[0..15].ProcessValue.SetPos := 0.0;
   softCam.cmAnodeMainPnP1AxisX.position[0..15].ProcessValue.inPos := FALSE;
   softCam.cmAnodeMainPnP1AxisX.position[0..15].ProcessValue.isBefore := FALSE;
   softCam.cmAnodeMainPnP1AxisX.position[0..15].ProcessValue.isAfter := FALSE;
   softCam.cmAnodeMainPnP1AxisX.position[0..15].ProcessValue.PosName := WSTRING#'';
   softCam.cmAnodeMainPnP1AxisY.TargetPosition := 0.0;
   softCam.cmAnodeMainPnP1AxisY.ActualPosition := 0.0;
   softCam.cmAnodeMainPnP1AxisY.UnitName := WSTRING#'';
   softCam.cmAnodeMainPnP1AxisY.error := FALSE;
   softCam.cmAnodeMainPnP1AxisY.status := 16#0000;
   softCam.cmAnodeMainPnP1AxisY.position[0..15].SetValue.Negative := 0.0;
   softCam.cmAnodeMainPnP1AxisY.position[0..15].SetValue.Postive := 0.0;
   softCam.cmAnodeMainPnP1AxisY.position[0..15].ProcessValue.Postive := 0.0;
   softCam.cmAnodeMainPnP1AxisY.position[0..15].ProcessValue.Negative := 0.0;
   softCam.cmAnodeMainPnP1AxisY.position[0..15].ProcessValue.SetPos := 0.0;
   softCam.cmAnodeMainPnP1AxisY.position[0..15].ProcessValue.inPos := FALSE;
   softCam.cmAnodeMainPnP1AxisY.position[0..15].ProcessValue.isBefore := FALSE;
   softCam.cmAnodeMainPnP1AxisY.position[0..15].ProcessValue.isAfter := FALSE;
   softCam.cmAnodeMainPnP1AxisY.position[0..15].ProcessValue.PosName := WSTRING#'';
   softCam.cmAnodeMainPnP1AxisZ.TargetPosition := 0.0;
   softCam.cmAnodeMainPnP1AxisZ.ActualPosition := 0.0;
   softCam.cmAnodeMainPnP1AxisZ.UnitName := WSTRING#'';
   softCam.cmAnodeMainPnP1AxisZ.error := FALSE;
   softCam.cmAnodeMainPnP1AxisZ.status := 16#0000;
   softCam.cmAnodeMainPnP1AxisZ.position[0..15].SetValue.Negative := 0.0;
   softCam.cmAnodeMainPnP1AxisZ.position[0..15].SetValue.Postive := 0.0;
   softCam.cmAnodeMainPnP1AxisZ.position[0..15].ProcessValue.Postive := 0.0;
   softCam.cmAnodeMainPnP1AxisZ.position[0..15].ProcessValue.Negative := 0.0;
   softCam.cmAnodeMainPnP1AxisZ.position[0..15].ProcessValue.SetPos := 0.0;
   softCam.cmAnodeMainPnP1AxisZ.position[0..15].ProcessValue.inPos := FALSE;
   softCam.cmAnodeMainPnP1AxisZ.position[0..15].ProcessValue.isBefore := FALSE;
   softCam.cmAnodeMainPnP1AxisZ.position[0..15].ProcessValue.isAfter := FALSE;
   softCam.cmAnodeMainPnP1AxisZ.position[0..15].ProcessValue.PosName := WSTRING#'';
   softCam.cmAnodeMainPnP2AxisX.TargetPosition := 0.0;
   softCam.cmAnodeMainPnP2AxisX.ActualPosition := 0.0;
   softCam.cmAnodeMainPnP2AxisX.UnitName := WSTRING#'';
   softCam.cmAnodeMainPnP2AxisX.error := FALSE;
   softCam.cmAnodeMainPnP2AxisX.status := 16#0000;
   softCam.cmAnodeMainPnP2AxisX.position[0..15].SetValue.Negative := 0.0;
   softCam.cmAnodeMainPnP2AxisX.position[0..15].SetValue.Postive := 0.0;
   softCam.cmAnodeMainPnP2AxisX.position[0..15].ProcessValue.Postive := 0.0;
   softCam.cmAnodeMainPnP2AxisX.position[0..15].ProcessValue.Negative := 0.0;
   softCam.cmAnodeMainPnP2AxisX.position[0..15].ProcessValue.SetPos := 0.0;
   softCam.cmAnodeMainPnP2AxisX.position[0..15].ProcessValue.inPos := FALSE;
   softCam.cmAnodeMainPnP2AxisX.position[0..15].ProcessValue.isBefore := FALSE;
   softCam.cmAnodeMainPnP2AxisX.position[0..15].ProcessValue.isAfter := FALSE;
   softCam.cmAnodeMainPnP2AxisX.position[0..15].ProcessValue.PosName := WSTRING#'';
   softCam.cmAnodeMainPnP2AxisZ.TargetPosition := 0.0;
   softCam.cmAnodeMainPnP2AxisZ.ActualPosition := 0.0;
   softCam.cmAnodeMainPnP2AxisZ.UnitName := WSTRING#'';
   softCam.cmAnodeMainPnP2AxisZ.error := FALSE;
   softCam.cmAnodeMainPnP2AxisZ.status := 16#0000;
   softCam.cmAnodeMainPnP2AxisZ.position[0..15].SetValue.Negative := 0.0;
   softCam.cmAnodeMainPnP2AxisZ.position[0..15].SetValue.Postive := 0.0;
   softCam.cmAnodeMainPnP2AxisZ.position[0..15].ProcessValue.Postive := 0.0;
   softCam.cmAnodeMainPnP2AxisZ.position[0..15].ProcessValue.Negative := 0.0;
   softCam.cmAnodeMainPnP2AxisZ.position[0..15].ProcessValue.SetPos := 0.0;
   softCam.cmAnodeMainPnP2AxisZ.position[0..15].ProcessValue.inPos := FALSE;
   softCam.cmAnodeMainPnP2AxisZ.position[0..15].ProcessValue.isBefore := FALSE;
   softCam.cmAnodeMainPnP2AxisZ.position[0..15].ProcessValue.isAfter := FALSE;
   softCam.cmAnodeMainPnP2AxisZ.position[0..15].ProcessValue.PosName := WSTRING#'';
   softCam.cmAnodeAlignTableAxisX.TargetPosition := 0.0;
   softCam.cmAnodeAlignTableAxisX.ActualPosition := 0.0;
   softCam.cmAnodeAlignTableAxisX.UnitName := WSTRING#'';
   softCam.cmAnodeAlignTableAxisX.error := FALSE;
   softCam.cmAnodeAlignTableAxisX.status := 16#0000;
   softCam.cmAnodeAlignTableAxisX.position[0..15].SetValue.Negative := 0.0;
   softCam.cmAnodeAlignTableAxisX.position[0..15].SetValue.Postive := 0.0;
   softCam.cmAnodeAlignTableAxisX.position[0..15].ProcessValue.Postive := 0.0;
   softCam.cmAnodeAlignTableAxisX.position[0..15].ProcessValue.Negative := 0.0;
   softCam.cmAnodeAlignTableAxisX.position[0..15].ProcessValue.SetPos := 0.0;
   softCam.cmAnodeAlignTableAxisX.position[0..15].ProcessValue.inPos := FALSE;
   softCam.cmAnodeAlignTableAxisX.position[0..15].ProcessValue.isBefore := FALSE;
   softCam.cmAnodeAlignTableAxisX.position[0..15].ProcessValue.isAfter := FALSE;
   softCam.cmAnodeAlignTableAxisX.position[0..15].ProcessValue.PosName := WSTRING#'';
   softCam.cmAnodeAlignTableAxisY1.TargetPosition := 0.0;
   softCam.cmAnodeAlignTableAxisY1.ActualPosition := 0.0;
   softCam.cmAnodeAlignTableAxisY1.UnitName := WSTRING#'';
   softCam.cmAnodeAlignTableAxisY1.error := FALSE;
   softCam.cmAnodeAlignTableAxisY1.status := 16#0000;
   softCam.cmAnodeAlignTableAxisY1.position[0..15].SetValue.Negative := 0.0;
   softCam.cmAnodeAlignTableAxisY1.position[0..15].SetValue.Postive := 0.0;
   softCam.cmAnodeAlignTableAxisY1.position[0..15].ProcessValue.Postive := 0.0;
   softCam.cmAnodeAlignTableAxisY1.position[0..15].ProcessValue.Negative := 0.0;
   softCam.cmAnodeAlignTableAxisY1.position[0..15].ProcessValue.SetPos := 0.0;
   softCam.cmAnodeAlignTableAxisY1.position[0..15].ProcessValue.inPos := FALSE;
   softCam.cmAnodeAlignTableAxisY1.position[0..15].ProcessValue.isBefore := FALSE;
   softCam.cmAnodeAlignTableAxisY1.position[0..15].ProcessValue.isAfter := FALSE;
   softCam.cmAnodeAlignTableAxisY1.position[0..15].ProcessValue.PosName := WSTRING#'';
   softCam.cmAnodeAlignTableAxisY2.TargetPosition := 0.0;
   softCam.cmAnodeAlignTableAxisY2.ActualPosition := 0.0;
   softCam.cmAnodeAlignTableAxisY2.UnitName := WSTRING#'';
   softCam.cmAnodeAlignTableAxisY2.error := FALSE;
   softCam.cmAnodeAlignTableAxisY2.status := 16#0000;
   softCam.cmAnodeAlignTableAxisY2.position[0..15].SetValue.Negative := 0.0;
   softCam.cmAnodeAlignTableAxisY2.position[0..15].SetValue.Postive := 0.0;
   softCam.cmAnodeAlignTableAxisY2.position[0..15].ProcessValue.Postive := 0.0;
   softCam.cmAnodeAlignTableAxisY2.position[0..15].ProcessValue.Negative := 0.0;
   softCam.cmAnodeAlignTableAxisY2.position[0..15].ProcessValue.SetPos := 0.0;
   softCam.cmAnodeAlignTableAxisY2.position[0..15].ProcessValue.inPos := FALSE;
   softCam.cmAnodeAlignTableAxisY2.position[0..15].ProcessValue.isBefore := FALSE;
   softCam.cmAnodeAlignTableAxisY2.position[0..15].ProcessValue.isAfter := FALSE;
   softCam.cmAnodeAlignTableAxisY2.position[0..15].ProcessValue.PosName := WSTRING#'';
END_DATA_BLOCK
